// TIA Portal V16 export
// export: Created 2024-05-10T06:46:45.0765115Z, ExportSetting WithDefaults, DisplayName Totally Integrated Automation Portal, DisplayVersion V16, DisplayName TIA Portal Version Control Interface, DisplayVersion V16, DisplayName TIA Portal Openness, DisplayVersion V16, DisplayName STEP 7 Professional, DisplayVersion V16, DisplayName STEP 7 Safety, DisplayVersion V16, DisplayName WinCC Professional, DisplayVersion V16
VAR_GLOBAL   // PLC tag table "103输入点变量表"
   EN_INV1故障 AT %I2.0 : Bool;
   Air故障 AT %I2.1 : Bool;
   EN_前端LS AT %I2.2 : Bool;
   EN_后端LS AT %I2.3 : Bool;
   EN_阻挡上升端 AT %I2.4 : Bool;
   EN_阻挡下降端 AT %I2.5 : Bool;
   EN_上升端 AT %I2.6 : Bool;
   EN_下降端 AT %I2.7 : Bool;
   EX_INV2故障 AT %I3.0 : Bool;
   干涉确认LS AT %I3.1 : Bool;
   EX_前端LS AT %I3.2 : Bool;
   EX_后端LS AT %I3.3 : Bool;
   EX_阻挡上升端 AT %I3.4 : Bool;
   EX_阻挡下降端 AT %I3.5 : Bool;
   EX_上升端 AT %I3.6 : Bool;
   EX_下降端 AT %I3.7 : Bool;
   ST01上层前端LS AT %I4.0 : Bool;
   ST01上层后端LS AT %I4.1 : Bool;
   ST01上阻挡上升端 AT %I4.2 : Bool;
   ST01上阻挡下降端 AT %I4.3 : Bool;
   ST01下层前端LS AT %I4.4 : Bool;
   ST01下层后端LS AT %I4.5 : Bool;
   ST01下阻挡上升端 AT %I4.6 : Bool;
   ST01下阻挡下降端 AT %I4.7 : Bool;
   ST02上层前端LS AT %I5.0 : Bool;
   ST02上层后端LS AT %I5.1 : Bool;
   ST02上阻挡上升端 AT %I5.2 : Bool;
   ST02上阻挡下降端 AT %I5.3 : Bool;
   ST02下层前端LS AT %I5.4 : Bool;
   ST02下层后端LS AT %I5.5 : Bool;
   ST02下阻挡上升端 AT %I5.6 : Bool;
   ST02下阻挡下降端 AT %I5.7 : Bool;
   ST03上层前端LS AT %I6.0 : Bool;
   ST03上层后端LS AT %I6.1 : Bool;
   ST03上阻挡上升端 AT %I6.2 : Bool;
   ST03上阻挡下降端 AT %I6.3 : Bool;
   ST03下层前端LS AT %I6.4 : Bool;
   ST03下层后端LS AT %I6.5 : Bool;
   ST03下阻挡上升端 AT %I6.6 : Bool;
   ST03下阻挡下降端 AT %I6.7 : Bool;
   ST04上层前端LS AT %I7.0 : Bool;
   ST04上层后端LS AT %I7.1 : Bool;
   ST04上阻挡上升端 AT %I7.2 : Bool;
   ST04上阻挡下降端 AT %I7.3 : Bool;
   ST05上层前端LS AT %I7.4 : Bool;
   ST05上层后端LS AT %I7.5 : Bool;
   ST05上阻挡上升端 AT %I7.6 : Bool;
   ST05上阻挡下降端 AT %I7.7 : Bool;
   前段_INV3故障 AT %I8.0 : Bool;
   前段_INV4故障 AT %I8.1 : Bool;
   后段_INV5故障 AT %I8.2 : Bool;
   后段_INV6故障 AT %I8.3 : Bool;
   ST06上层前端LS AT %I8.4 : Bool;
   ST06上层后端LS AT %I8.5 : Bool;
   ST06上阻挡上升端 AT %I8.6 : Bool;
   ST06上阻挡下降端 AT %I8.7 : Bool;
   ST07上层前端LS AT %I9.0 : Bool;
   ST07上层后端LS AT %I9.1 : Bool;
   ST07上阻挡上升端 AT %I9.2 : Bool;
   ST07上阻挡下降端 AT %I9.3 : Bool;
   ST08上层前端LS AT %I9.4 : Bool;
   ST08上层后端LS AT %I9.5 : Bool;
   ST08上阻挡上升端 AT %I9.6 : Bool;
   ST08上阻挡下降端 AT %I9.7 : Bool;
   ST09上层前端LS AT %I10.0 : Bool;
   ST09上层后端LS AT %I10.1 : Bool;
   ST09上阻挡上升端 AT %I10.2 : Bool;
   ST09上阻挡下降端 AT %I10.3 : Bool;
   ST10上层前端LS AT %I10.4 : Bool;
   ST10上层后端LS AT %I10.5 : Bool;
   ST10上阻挡上升端 AT %I10.6 : Bool;
   ST10上阻挡下降端 AT %I10.7 : Bool;
   ST11上层前端LS AT %I11.0 : Bool;
   ST11上层后端LS AT %I11.1 : Bool;
   ST11上阻挡上升端 AT %I11.2 : Bool;
   ST11上阻挡下降端 AT %I11.3 : Bool;
   ST12上层前端LS AT %I11.4 : Bool;
   ST12上层后端LS AT %I11.5 : Bool;
   ST12上阻挡上升端 AT %I11.6 : Bool;
   ST12上阻挡下降端 AT %I11.7 : Bool;
   ST01急停EM AT %I12.0 : Bool;
   ST01放行SB AT %I12.1 : Bool;
   ST02急停EM AT %I12.2 : Bool;
   ST02放行SB AT %I12.3 : Bool;
   ST03急停EM AT %I12.4 : Bool;
   ST03放行SB AT %I12.5 : Bool;
   ST04急停EM AT %I12.6 : Bool;
   ST04放行SB AT %I12.7 : Bool;
   ST05急停EM AT %I13.0 : Bool;
   ST05放行SB AT %I13.1 : Bool;
   ST06急停EM AT %I13.2 : Bool;
   ST06放行SB AT %I13.3 : Bool;
   ST07急停EM AT %I14.0 : Bool;
   ST07放行SB AT %I14.1 : Bool;
   ST08急停EM AT %I14.2 : Bool;
   ST08放行SB AT %I14.3 : Bool;
   ST09急停EM AT %I14.4 : Bool;
   ST09放行SB AT %I14.5 : Bool;
   ST10急停EM AT %I14.6 : Bool;
   ST10放行SB AT %I14.7 : Bool;
   ST11急停EM AT %I15.0 : Bool;
   ST11放行SB AT %I15.1 : Bool;
   ST12急停EM AT %I15.2 : Bool;
   ST12放行SB AT %I15.3 : Bool;
END_VAR
